INTERFACE I_Sequenz

METHOD M_Start : BOOL
VAR_INPUT
END_VAR
END_METHOD

METHOD M_Stop : BOOL
VAR_INPUT
END_VAR
END_METHOD

PROPERTY P_Finished : BOOL;
GET
END_GET
END_PROPERTY

END_INTERFACE

(* stored: Version 1.1.0.1
   Itf I_Sequenz: Id {dbc39906-6275-4e7d-8de7-806828a808dc}
   Method M_Start: Id {3f503f57-3734-4ad6-8d87-517dc605a09e}
   Method M_Stop: Id {6a84f33b-01aa-4820-b114-16013ce892bf}
   Property P_Finished: Id {eb901849-fec2-4cf4-98f9-fad5290e4c0f}
   Get Get: Id {410229d3-4f33-4850-9625-8c82b5fc1174} *)
